FUNCTION_BLOCK DSCYL_DIAGL (* Locally Coupled and Clocked Diagnostics for a Dual-Stroke Cylinder *)
  (* Standard: 61499-1; Classification: Diagnostics; ApplicationDomain: Mechanisms *)
  (* Version 0.2, 2005-06-01, JHC, Holobloc Inc, Re-compiled with new emitter. *)
  (* Version 0.1, 2004-10-21, JHC, Rockwell Automation, Renamed from DSCYL_DIAGCL. *)
  (* Version 0.0, 2004-08-14, JHC, Rockwell Automation *)
  (* Compiler header: package fb.rt.mach; import fb.rt.mva.*; import fb.rt.net.*; import fb.rt.math.*; *)
  (* Compiler classdef: public class DSCYL_DIAGL extends FBMVCD *)
  (* Compiler Java Sun JDK 1.4.2 *)
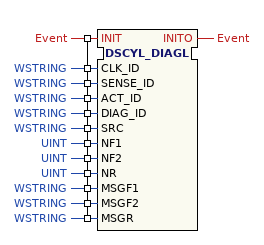
  EVENT_INPUT
    INIT WITH SENSE_ID, ACT_ID, DIAG_ID, SRC, NF1, NF2, NR, MSGF1, MSGF2, MSGR, CLK_ID;
  END_EVENT
  EVENT_OUTPUT
    INITO;
  END_EVENT
  VAR_INPUT
    CLK_ID : WSTRING := "DIAG_CLK"; (* Diagnostic Clock Local Channel ID *)
    SENSE_ID : WSTRING; (* Sensor channel ID from Model *)
    ACT_ID : WSTRING; (* Actuator channel ID from Controller *)
    DIAG_ID : WSTRING; (* Diagnostic output channel ID *)
    SRC : WSTRING; (* Diagnostic Source ID *)
    NF1 : UINT; (* Cylinder 1 Forward Motion Timeout Period in CLK cycles *)
    NF2 : UINT; (* Cylinder 2 Motion Timeout Period in CLK cycles *)
    NR : UINT; (* Reverse Motion Timeout Period in CLK cycles *)
    MSGF1 : WSTRING := "TIMEOUT_ADVANCING1"; (* Message for fault on forward motion of Cylinder 1 *)
    MSGF2 : WSTRING := "TIMEOUT_ADVANCING2"; (* Message for fault on forward motion of Cylinder 2 *)
    MSGR : WSTRING := "TIMEOUT_RETRACTING"; (* Message for fault on combined reverse motion *)
  END_VAR
  FBS
    ACT : SUBL_3;
    SENSE : SUBL_3;
    MONF1 : MECH1_DIAGL; (* Monitor Cylinder 1 Forward Motion *)
    MONF2 : MECH1_DIAGL; (* Monitor Cylinder 2 Forward motion *)
    MONR : MECH1_DIAGL; (* Monitor Reverse Motion of both cylinders *)
    NOT_F2 : FB_NOT;
    AND_F1 : FB_AND;
  END_FBS
  EVENT_CONNECTIONS
    MONF1.INITO TO MONF2.INIT;
    NOT_F2.CNF TO AND_F1.REQ;
    INIT TO ACT.INIT;
    SENSE.INITO TO MONF1.INIT;
    ACT.IND TO NOT_F2.REQ;
    ACT.INITO TO MONR.INIT;
    MONR.INITO TO SENSE.INIT;
    MONF2.INITO TO INITO;
  END_CONNECTIONS
  DATA_CONNECTIONS
    ACT_ID TO ACT.ID;
    SENSE_ID TO SENSE.ID;
    ACT.RD_2 TO MONF2.FWD;
    ACT.RD_3 TO MONR.FWD;
    SENSE.RD_1 TO MONR.END;
    SENSE.RD_2 TO MONF1.END;
    SENSE.RD_3 TO MONF2.END;
    CLK_ID TO MONF1.CLK_ID;
    DIAG_ID TO MONF1.DIAG_ID;
    NF1 TO MONF1.N;
    SRC TO MONF1.SRC;
    MSGF1 TO MONF1.MSG;
    CLK_ID TO MONF2.CLK_ID;
    DIAG_ID TO MONF2.DIAG_ID;
    NF2 TO MONF2.N;
    SRC TO MONF2.SRC;
    MSGF2 TO MONF2.MSG;
    NR TO MONR.N;
    SRC TO MONR.SRC;
    MSGR TO MONR.MSG;
    AND_F1.OUT TO MONF1.FWD;
    ACT.RD_2 TO NOT_F2.IN;
    ACT.RD_1 TO AND_F1.IN2;
    CLK_ID TO MONR.CLK_ID;
    DIAG_ID TO MONR.DIAG_ID;
    NOT_F2.OUT TO AND_F1.IN1;
  END_CONNECTIONS
END_FUNCTION_BLOCK
